FUNCTION_BLOCK FB_MotionDrive IMPLEMENTS I_MotionDrive
VAR_INPUT
END_VAR
VAR_OUTPUT
END_VAR
VAR
    stMotionDrive : ST_MotionDrive;
    stMotionEpicsInterface : ST_MotionEpicsInterface;

    iMotionAxis : I_MotionAxis;
    iBrake :I_Brake;
    iMotionInterlocks: I_MotionInterlocks;
    iMotionLogger : I_MotionLogger;
    iPersistantDataStorage : I_PersistantDataStorage;

END_VAR

THIS^.NCParamsExposed();

{warning 'Add property implementation'}
PROPERTY Error : BOOL
GET
END_GET
SET
END_SET
END_PROPERTY

{warning 'Add property implementation'}
PROPERTY ErrorCode : UDINT
GET
END_GET
SET
END_SET
END_PROPERTY

//FB_Init is always available implicitly and it is used primarily for initialization.
//The return value is not evaluated. For a specific influence, you can also declare the
//methods explicitly and provide additional code there with the standard initialization
//code. You can evaluate the return value.
METHOD FB_Init: BOOL
VAR_INPUT
    bInitRetains: BOOL; // TRUE: the retain variables are initialized (reset warm / reset cold)
    bInCopyCode: BOOL;  // TRUE: the instance will be copied to the copy code afterward (online change)
    //Declaration
    iMotionAxis: I_MotionAxis;
    iBrake : I_Brake;
    iMotionInterlocks : I_MotionInterlocks;
    iMotionLogger : I_MotionLogger;
    iPersistantDataStorage: I_PersistantDataStorage;
END_VAR
// Body
THIS^.iMotionAxis:=iMotionAxis;
THIS^.iBrake:=iBrake;
THIS^.iMotionInterlocks:=iMotionInterlocks;
THIS^.iPersistantDataStorage:=iPersistantDataStorage;
END_METHOD

{warning 'Add method implementation '}
METHOD GetInterlocksRef
END_METHOD

{warning 'Add method implementation '}
METHOD GetLoggerRef : REFERENCE TO AXIS_REF
END_METHOD

{warning 'Add method implementation '}
METHOD GetPersistantStorageRef
END_METHOD

{warning 'Add method implementation '}
METHOD HomeCmd
END_METHOD

{warning 'Add method implementation '}
METHOD MoveAbsolute
VAR_INPUT
    Position	: LREAL;
    Velocity	: LREAL;
    Acceleration	: LREAL := 0.0;
    Deceleration	: LREAL := 0.0;
    Jerk	: LREAL := 0.0;
    BufferMode	: MC_BufferMode := .MC_BufferMode.MC_Aborting;
END_VAR
VAR_OUTPUT
    Done	: BOOL;
    Busy	: BOOL;
    Active	: BOOL;
    CommandAborted	: BOOL;
    Error	: BOOL;
    ErrorID	: UDINT;
    ErrorStr	: T_MaxString;
END_VAR
END_METHOD

{warning 'Add method implementation '}
METHOD MoveCmd
END_METHOD

METHOD PROTECTED NCParamsExposed
VAR_INPUT
END_VAR
// Copy axis parameters that we want to expose to the EPICS layer.
stMotionEpicsInterface.stAxisParametersExposed.bCtrlEnablePosDiffControl     := iMotionAxis.CtrlEnablePosDiffControl;
stMotionEpicsInterface.stAxisParametersExposed.bEncEnableSoftEndMaxControl   := iMotionAxis.EncEnableSoftEndMaxControl;
stMotionEpicsInterface.stAxisParametersExposed.bEncEnableSoftEndMinControl   := iMotionAxis.EncEnableSoftEndMinControl;
stMotionEpicsInterface.stAxisParametersExposed.fAccelerationMax              := iMotionAxis.AccelerationMax;
stMotionEpicsInterface.stAxisParametersExposed.fCtrlPosDiffMax               := iMotionAxis.CtrlPosDiffMax;
stMotionEpicsInterface.stAxisParametersExposed.fCtrlPosDiffMaxTime           := iMotionAxis.CtrlPosDiffMaxTime;
stMotionEpicsInterface.stAxisParametersExposed.fDecelerationMax              := iMotionAxis.DecelerationMax;
stMotionEpicsInterface.stAxisParametersExposed.fEncSoftEndMax                := iMotionAxis.EncSoftEndMax;
stMotionEpicsInterface.stAxisParametersExposed.fEncSoftEndMin                := iMotionAxis.EncSoftEndMin;
stMotionEpicsInterface.stAxisParametersExposed.fVeloMaximum                  := iMotionAxis.VeloMaximum;
stMotionEpicsInterface.stAxisParametersExposed.fEncOffset               	 := iMotionAxis.EncOffset;
stMotionEpicsInterface.stAxisParametersExposed.fEncScaleFactorInternal       := iMotionAxis.EncScaleFactorInternal;

stMotionDrive.bAxisParamsInit S= iMotionAxis.NCParamsReadDone;
END_METHOD

{warning 'Add method implementation '}
METHOD ProcessMoveReq
END_METHOD

END_FUNCTION_BLOCK

(* stored: Version 1.1.0.1
   POU FB_MotionDrive: Id {ab485b6e-0ea0-46c8-a998-93ea4aaa54b4}, SpecialFunc None
   Property Error: Id {9e9f8ffe-6e96-4b18-9522-dd45ebc471b8}
   Get Get: Id {06a27d70-70de-4b99-a912-9d5fb421aef2}
   Set Set: Id {ec338d56-3b79-4ff9-ae9f-e315a8d5ee7f}
   Property ErrorCode: Id {82d12daf-7c03-42c7-91e0-028740989fb2}
   Get Get: Id {745866a5-7830-470f-94c1-1c5eacda59a5}
   Set Set: Id {b393c613-5b8a-4252-96ef-ba4124ed098d}
   Method FB_init: Id {15f40a72-aeff-42da-b103-42138a2002e8}
   Method GetInterlocksRef: Id {519cf572-57b6-4265-8a35-8e40f4725969}
   Method GetLoggerRef: Id {52d12a63-003f-46aa-9d7c-0766b0dbebaf}
   Method GetPersistantStorageRef: Id {0848ae24-3e4a-427c-bd3d-72c635281586}
   Method HomeCmd: Id {5473fbf2-fdd8-4d41-a230-673673ab7612}
   Method MoveAbsolute: Id {bcd9f3a9-147c-469e-8034-f278929d33ca}
   Method MoveCmd: Id {782b2d9d-6d1e-427f-8acb-bccc3e3fc3bb}
   Method NCParamsExposed: Id {a32b8f9b-a550-4cf6-9dc3-5c1e587d0657}
   Method ProcessMoveReq: Id {1da2dc9d-4406-4cb4-be2e-a29a35f201c7} *)
